Staubli VAL3: PROG.pjx

--- PROG.pjx ---
Parameters version=s7.5.3 stackSize=5000 millimeterUnit=true
Data file=PROG.dtx
Type name=InstrItem path=Disk://kernel/template/InstrItem/InstrItem.pjx
Type name=progItem path=Disk://kernel/template/progItem/progItem.pjx

--- PROG.dtx ---
public progItem pProg{}
  [HOME1]
    InstrItem iEvent
      [0]
        string sType
        string sData
    string sID = "HOME1"
  [HOME2]
    InstrItem iEvent
      [0]
        string sType
        string sData
    string sID = "HOME2"
